(* CoDeSys 2.3.9.48 project: Hausautomation.pro *)
(* Libraries: WagoBuilding_01.lib 14.9.16 07:36:54, SysLibRtc.lib 8.11.10 11:37:48, Gebaeude_allgemein.lib 16.4.15 11:31:36, SysLibTime.lib 8.11.10 11:37:48, Standard.lib*2.6.14 10:37:46, SYSLIBCALLBACK.LIB 8.11.10 11:37:48, Iecsfc.lib 2.6.14 10:37:46 *)

(* PLC configuration (modules and I/O channels)
KA01_KL01_DI AT %IX0.0 [BOOLOnX_I] 1: Flur OG 1 (unten) (Dach 2)
KA01_KL02_DI AT %IX0.1 [BOOLOnX_I] 2: Treppe EG 1
KA02_KL01_DI AT %IX0.2 [BOOLOnX_I] 3: Büro Tür
KA02_KL02_DI AT %IX0.3 [BOOLOnX_I] 4: Eltern Tür
KA02_KL03_DI AT %IX0.4 [BOOLOnX_I] 5: Kind Tür
KA02_KL04_DI AT %IX0.5 [BOOLOnX_I] 6: Küche Tür
KA02_KL05_DI AT %IX0.6 [BOOLOnX_I] 7: WZ Flurtür 1
KA02_KL06_DI AT %IX0.7 [BOOLOnX_I] 8: WZ Terassentür 1
KA02_KL07_DI AT %IX0.8 [BOOLOnX_I] 9: WZ Flurtür 2
KA02_KL08_DI AT %IX0.9 [BOOLOnX_I] 10: Flur Tür WZ
0750-0430 8 DI 24 V DC 3.0ms [Type_1_8_Channels] node 2, in %IX0.2 out %QB0 {INTTypePAAssignment = PLC; INTTypeModule = plugged}
  KA03_KL01_DI AT %IX0.10 [BOOLOnX_I] 11: WZ groß up
  KA03_KL02_DI AT %IX0.11 [BOOLOnX_I] 12: WZ groß: down
  KA03_KL03_DI AT %IX0.12 [BOOLOnX_I] 13: WZ klein up
  KA03_KL04_DI AT %IX0.13 [BOOLOnX_I] 14: WZ klein down
  KA03_KL05_DI AT %IX0.14 [BOOLOnX_I] 15: Kind up
  KA03_KL06_DI AT %IX0.15 [BOOLOnX_I] 16: Kind down
  KA03_KL07_DI AT %IX1.0 [BOOLOnX_I] 17: WZ Tür up
  KA03_KL08_DI AT %IX1.1 [BOOLOnX_I] 18: WZ Tür down
  KA04_KL01_DI AT %IX1.2 [BOOLOnX_I] 19: Eltern down
  KA04_KL02_DI AT %IX1.3 [BOOLOnX_I] 20: Eltern up
  KA04_KL03_DI AT %IX1.4 [BOOLOnX_I] 21: Treppe EG 2
  KA04_KL04_DI AT %IX1.5 [BOOLOnX_I] 22: Haustür
  KA04_KL05_DI AT %IX1.6 [BOOLOnX_I] 23: Flur OG 2 (oben) (Dach 2)
  KA04_KL06_DI AT %IX1.7 [BOOLOnX_I] 24: WZ Flurtür2
  KA04_KL07_DI AT %IX1.8 [BOOLOnX_I] 25: Wand WZ
  KA04_KL08_DI AT %IX1.9 [BOOLOnX_I] 26: Dach Taster 1
KA05_KL01_DO AT %QX0.0 [BOOLOnX_Q] 1: Flur OG
KA05_KL02_DO AT %QX0.1 [BOOLOnX_Q] 2: Flur EG
KA06_KL01_DO AT %QX0.2 [BOOLOnX_Q] 3: Büro
KA06_KL02_DO AT %QX0.3 [BOOLOnX_Q] 4: Eltern
KA06_KL03_DO AT %QX0.4 [BOOLOnX_Q] 5: Kind
KA06_KL04_DO AT %QX0.5 [BOOLOnX_Q] 6: Küche
KA06_KL05_DO AT %QX0.6 [BOOLOnX_Q] 7: WZ 1
KA06_KL06_DO AT %QX0.7 [BOOLOnX_Q] 8: WZ 2
KA06_KL07_DO AT %QX0.8 [BOOLOnX_Q] 9: Essecke Steckdose 1
KA06_KL08_DO AT %QX0.9 [BOOLOnX_Q] 10: Essecke Steckdose 2
KA07_KL01_DO AT %QX0.10 [BOOLOnX_Q] 11: WZ groß down
KA07_KL02_DO AT %QX0.11 [BOOLOnX_Q] 12: WZ groß up
KA07_KL03_DO AT %QX0.12 [BOOLOnX_Q] 13: WZ klein up
KA07_KL04_DO AT %QX0.13 [BOOLOnX_Q] 14: WZ klein down
KA07_KL05_DO AT %QX0.14 [BOOLOnX_Q] 15: Kind down
KA07_KL06_DO AT %QX0.15 [BOOLOnX_Q] 16: Kind up
KA07_KL07_DO AT %QX1.0 [BOOLOnX_Q] 17: Eltern up
KA07_KL08_DO AT %QX1.1 [BOOLOnX_Q] 18: Eltern down
KA08_KL01_DO AT %QX1.2 [BOOLOnX_Q] 19: WZ Tür down
KA08_KL02_DO AT %QX1.3 [BOOLOnX_Q] 20: WZ Tür up
KA08_KL03_DO AT %QX1.4 [BOOLOnX_Q] 21: Dach Lampe 1
KA08_KL04_DO AT %QX1.5 [BOOLOnX_Q] 22: Treppenhaus OG LEDs
KA08_KL05_DO AT %QX1.6 [BOOLOnX_Q] 23: -
KA08_KL06_DO AT %QX1.7 [BOOLOnX_Q] 24: -
KA08_KL07_DO AT %QX1.8 [BOOLOnX_Q] 25: Dach Licht 1
KA08_KL08_DO AT %QX1.9 [BOOLOnX_Q] 26: Dach Licht 2
KA09_KL01_DI AT %IX1.10 [BOOLOnX_I] 27: WZ Terassentür 2
KA09_KL02_DI AT %IX1.11 [BOOLOnX_I] 28: WZ Terassentür 3
KA09_KL03_DI AT %IX1.12 [BOOLOnX_I] 29: WZ Terassentür 4
KA09_KL04_DI AT %IX1.13 [BOOLOnX_I] 30: Büro Up
KA09_KL05_DI AT %IX1.14 [BOOLOnX_I] 31: Büro Down
KA09_KL06_DI AT %IX1.15 [BOOLOnX_I] 32: Küche Down
KA09_KL07_DI AT %IX2.0 [BOOLOnX_I] 33: Küche Up
KA09_KL08_DI AT %IX2.1 [BOOLOnX_I] 34: Dach Taster 2
KA10_KL01_DO AT %QX1.10 [BOOLOnX_Q] 35: Küche Down
KA10_KL02_DO AT %QX1.11 [BOOLOnX_Q] 36: Büro Up
KA10_KL03_DO AT %QX1.12 [BOOLOnX_Q] 37: Büro Down
KA10_KL04_DO AT %QX1.13 [BOOLOnX_Q] 38: Küche Up
KA10_KL05_DO AT %QX1.14 [BOOLOnX_Q] Ch_5 Digital output
KA10_KL06_DO AT %QX1.15 [BOOLOnX_Q] Ch_6 Digital output
KA10_KL07_DO AT %QX2.0 [BOOLOnX_Q] Ch_7 Digital output
KA10_KL08_DO AT %QX2.1 [BOOLOnX_Q] Ch_8 Digital output
KA10_KL09_DO AT %QX2.2 [BOOLOnX_Q] Ch_9 Digital output
KA10_KL10_DO AT %QX2.3 [BOOLOnX_Q] Ch_10 Digital output
KA10_KL11_DO AT %QX2.4 [BOOLOnX_Q] Ch_11 Digital output
KA10_KL12_DO AT %QX2.5 [BOOLOnX_Q] Ch_12 Digital output
KA10_KL13_DO AT %QX2.6 [BOOLOnX_Q] Ch_13 Digital output
KA10_KL14_DO AT %QX2.7 [BOOLOnX_Q] Ch_14 Digital output
KA10_KL15_DO AT %QX2.8 [BOOLOnX_Q] Ch_15 Digital output
KA10_KL16_DO AT %QX2.9 [BOOLOnX_Q] Ch_16 Digital output
Fieldbus variables [FB_VARS] node 1, in %IB0 out %QB0
BOOL, Flag [FLAG_BOOL] node 1, in %IB0 out %QB0
  LichtFlurEG AT %MX0.0 [BOOLOnX_Q] LichtFlurEG(Ausgang)
BOOL, Flag [FLAG_BOOL] node 2, in %IB0 out %QB0
  LichtWohnzimmer AT %MX0.1 [BOOLOnX_Q] LichtWohnzimmer(Ausgang)
BOOL, Flag [FLAG_BOOL] node 3, in %IB0 out %QB0
  LichtKueche AT %MX0.2 [BOOLOnX_Q] LichtKueche(Ausgang)
BOOL, Flag [FLAG_BOOL] node 4, in %IB0 out %QB0
  LichtStehlampe AT %MX0.3 [BOOLOnX_Q] LichtStehlampe(Ausgang)
BOOL, Flag [FLAG_BOOL] node 5, in %IB0 out %QB0
  LichtBuero AT %MX0.4 [BOOLOnX_Q] LichtBuero(Ausgang)
BOOL, Flag [FLAG_BOOL] node 6, in %IB0 out %QB0
  LichtSchlafzimmer AT %MX0.5 [BOOLOnX_Q] LichtSchlafzimmer(Ausgang)
BOOL, Flag [FLAG_BOOL] node 7, in %IB0 out %QB0
  LichtAnnika AT %MX0.6 [BOOLOnX_Q] LichtAnnika(Ausgang)
BOOL, Flag [FLAG_BOOL] node 8, in %IB0 out %QB0
  LichtFlurOG AT %MX0.7 [BOOLOnX_Q] LichtFlurOG(Ausgang)
BOOL, Flag [FLAG_BOOL] node 9, in %IB0 out %QB0
  TasterBuero AT %MX0.8 [BOOLOnX_Q] TasterBuero(Eingang)
BOOL, Flag [FLAG_BOOL] node 10, in %IB0 out %QB0
  TasterFlurEG AT %MX0.9 [BOOLOnX_Q] TasterFlurEG(Eingang)
BOOL, Flag [FLAG_BOOL] node 11, in %IB0 out %QB0
  TasterWohnzimmer AT %MX0.10 [BOOLOnX_Q] TasterWohnzimmer(Eingang)
BOOL, Flag [FLAG_BOOL] node 12, in %IB0 out %QB0
  TasterKueche AT %MX0.11 [BOOLOnX_Q] TasterKueche(Eingang)
BOOL, Flag [FLAG_BOOL] node 13, in %IB0 out %QB0
  TasterStehlampe AT %MX0.12 [BOOLOnX_Q] TasterStehlampe(Eingang)
BOOL, Flag [FLAG_BOOL] node 14, in %IB0 out %QB0
  TasterSchlafzimmer AT %MX0.13 [BOOLOnX_Q] TasterSchlafzimmer(Eingang)
BOOL, Flag [FLAG_BOOL] node 15, in %IB0 out %QB0
  TasterAnnika AT %MX0.14 [BOOLOnX_Q] TasterAnnika(Eingang)
BOOL, Flag [FLAG_BOOL] node 16, in %IB0 out %QB0
  TasterFlurOG AT %MX0.15 [BOOLOnX_Q] TasterFlurOG(Eingang)
BOOL, Flag [FLAG_BOOL] node 17, in %IB0 out %QB0
  JalousieElternUp AT %MX1.0 [BOOLOnX_Q] Jalousie Eltern Hoch
BOOL, Flag [FLAG_BOOL] node 18, in %IB0 out %QB0
  JalousieElternDown AT %MX1.1 [BOOLOnX_Q] Jalousie Eltern Runter
BOOL, Flag [FLAG_BOOL] node 19, in %IB0 out %QB0
  JalousieAnnikaDown AT %MX1.2 [BOOLOnX_Q] Jalousie Annika runter
BOOL, Flag [FLAG_BOOL] node 20, in %IB0 out %QB0
  JalousieAnnikaUp AT %MX1.3 [BOOLOnX_Q] Jalousie Annika hoch
BOOL, Flag [FLAG_BOOL] node 21, in %IB0 out %QB0
  JalousieWohnzimmerGrossDown AT %MX1.4 [BOOLOnX_Q] Jalousie Wohnzimmer großes Fenster runter
BOOL, Flag [FLAG_BOOL] node 22, in %IB0 out %QB0
  JalousieWohnzimmerGrossUp AT %MX1.5 [BOOLOnX_Q] Jalousie Wohnzimmer großes Fenster hoch
BOOL, Flag [FLAG_BOOL] node 23, in %IB0 out %QB0
  JalousieWohnzimmerTuerDown AT %MX1.6 [BOOLOnX_Q] Jalousie Wohnzimmer Tür runter
BOOL, Flag [FLAG_BOOL] node 24, in %IB0 out %QB0
  JalousieWohnzimmerTuerUp AT %MX1.7 [BOOLOnX_Q] Jalousie Wohnzimmer Tür hoch
BOOL, Flag [FLAG_BOOL] node 25, in %IB0 out %QB0
  JalousieWohnzimmerKleinDown AT %MX1.8 [BOOLOnX_Q] Jalousie Wohnzimmer kleines Fenster runter
BOOL, Flag [FLAG_BOOL] node 26, in %IB0 out %QB0
  JalousieWohnzimmerKleinUp AT %MX1.9 [BOOLOnX_Q] Jalousie Wohnzimmer kleines Fenster hoch
BOOL, Flag [FLAG_BOOL] node 27, in %IB0 out %QB0
  JalousieBueroUp AT %MX1.10 [BOOLOnX_Q] Jalousie Büro hoch
BOOL, Flag [FLAG_BOOL] node 28, in %IB0 out %QB0
  JalousieBueroDown AT %MX1.11 [BOOLOnX_Q] Jalousie Büro runter
BOOL, Flag [FLAG_BOOL] node 29, in %IB0 out %QB0
  JalousieKuecheUp AT %MX1.12 [BOOLOnX_Q] Jalousie Küche hoch
BOOL, Flag [FLAG_BOOL] node 30, in %IB0 out %QB0
  JalousieKuecheDown AT %MX1.13 [BOOLOnX_Q] Jalousie Küche runter
BOOL, Flag [FLAG_BOOL] node 31, in %IB0 out %QB0
  TasterLichtDachboden AT %MX1.14 [BOOLOnX_Q] Taster Licht Dachboden
BOOL, Flag [FLAG_BOOL] node 32, in %IB0 out %QB0
  LichtDachbodenVorne AT %MX1.15 [BOOLOnX_Q] Licht Dachboden vorne (Büro)
BOOL, Flag [FLAG_BOOL] node 33, in %IB0 out %QB0
  LichtDachbodenHinten AT %MX2.0 [BOOLOnX_Q] Licht Dachboden hinten (Gästezimmer)
Modbus-Master [MB_MASTER] node 3, in %IB0 out %QB0
*)

(* Task configuration *)
TASK MAIN (PRIORITY := 1, INTERVAL := T#200ms);
	PLC_PRG();
END_TASK

(* Global variable list: Globale_Variablen *)
VAR_GLOBAL

	LIGHT_CentralOn: BOOL := FALSE;
	LIGHT_CentralOff: BOOL := FALSE;
	WZ_2_AN: BOOL;

	YEAR: WORD;
	MONTH: BYTE;
	DAY: BYTE;
	HOUR: BYTE;
	MINUTE: BYTE;
	SECOND: BYTE;
	WEEK_DAY: BYTE;


      DAY_BOOL: BOOL;
      NIGHT_BOOL: BOOL;

	BLINDS_CentralUp: BOOL := FALSE;
	BLINDS_LfzGesamt: UINT := 700;
	BLINDS_PauseAufAb: UINT := 5;
	BLINDS_TasKurz: UINT := 5;
	BLINDS_LfzBeschattPos: UINT := 10;
	BLINDS_LfzKurz: UINT := 400;
	BLINDS_WendeZeitLamelle: UINT := 40;
END_VAR

(* POU PLC_PRG, ST *)
PROGRAM PLC_PRG
LIGHTS_FLUR_EG;
LIGHTS_FLUR_OG;
LIGHTS_WZ;
LIGHTS_KUECHE;
LIGHTS_BUERO;
LIGHTS_SCHLAFZIMMER;
LIGHTS_ANNIKA;
LIGHTS_STEHLAMPE;
LIGHTS_DRAUSSEN;
UHRZEIT;
BLINDS_WZ;
BLINDS_ANNIKA;
BLINDS_ELTERN;
BLINDS_BUERO;
BLINDS_KUECHE;
LIGHTS_ATTIC;
IsDay;
END_PROGRAM

(* POU LIGHTS_FLUR_EG, CFC *)
PROGRAM LIGHTS_FLUR_EG
VAR
	FB_LIGHT_02: FbLatchedRelay;
	F_Treppe_1: F_TRIG;
	F_Treppe_2: R_TRIG;
	FB_LIGHT_02_2: FbLatchedRelay;
	F_Haustuer_1: F_TRIG;
	F_Haustuer_2: R_TRIG;
	F_FlurTuerWZ_1: F_TRIG;
	F_FlurTuerWZ_2: R_TRIG;
	F_Flur_oben_1: F_TRIG;
	F_Flur_oben_2: R_TRIG;
	F_Flur_OG_1: F_TRIG;
	F_Flur_OG_2: R_TRIG;
	F_Flur_EG_5: F_TRIG;
	F_Flur_EG_6: R_TRIG;
	F_Flur_EG_openhab: F_TRIG;
	F_Flur_openhab: R_TRIG;
	R_Flur_EG_openhab: R_TRIG;
END_VAR
VAR (* helpers for the ST form of the networks *)
	_t138 : BOOL;
END_VAR
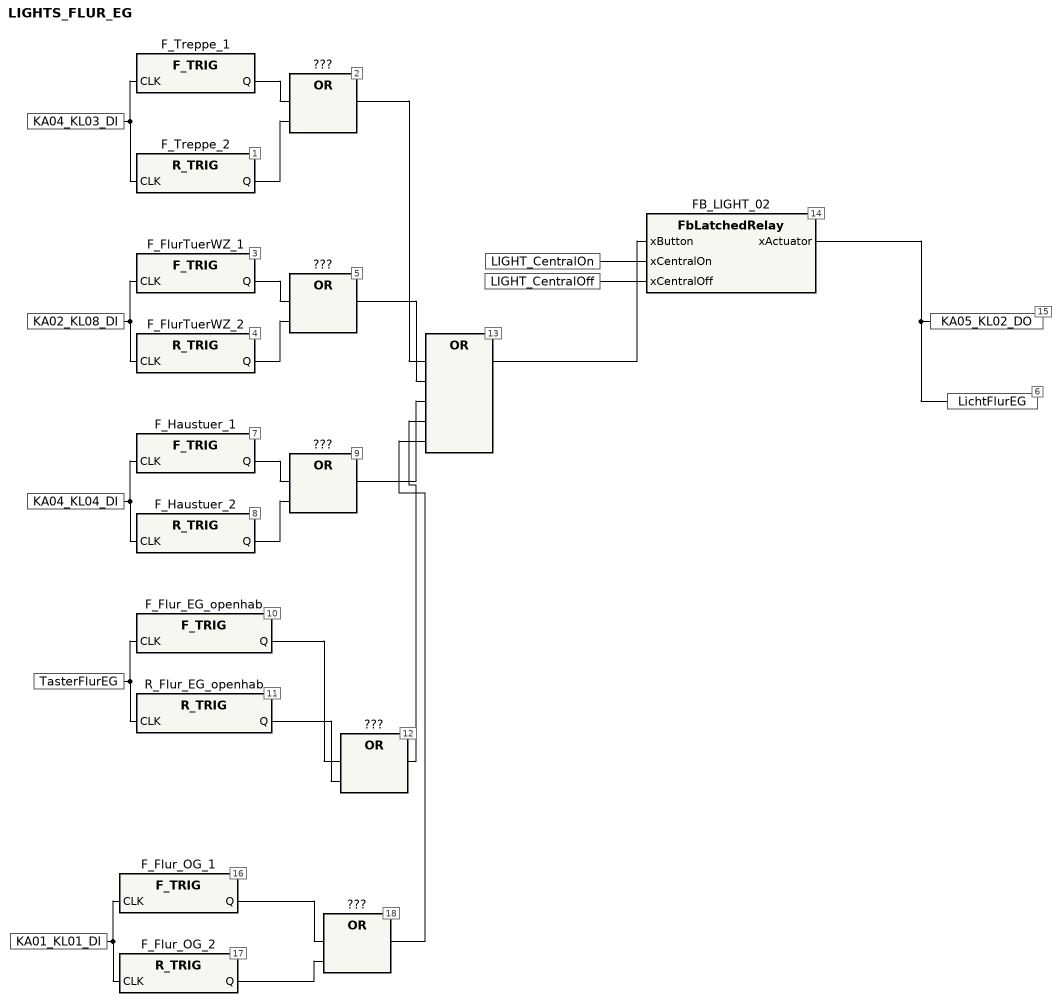
_CFC_ (* Continuous Function Chart, elements in execution order *)
#0 F_Treppe_1:F_TRIG(CLK: KA04_KL03_DI)
#1 F_Treppe_2:R_TRIG(CLK: KA04_KL03_DI)
#2 ???:OR(#0.Q, #1.Q)
#3 F_FlurTuerWZ_1:F_TRIG(CLK: KA02_KL08_DI)
#4 F_FlurTuerWZ_2:R_TRIG(CLK: KA02_KL08_DI)
#5 ???:OR(#3.Q, #4.Q)
#6 LichtFlurEG <= #14.xActuator
#7 F_Haustuer_1:F_TRIG(CLK: KA04_KL04_DI)
#8 F_Haustuer_2:R_TRIG(CLK: KA04_KL04_DI)
#9 ???:OR(#7.Q, #8.Q)
#10 F_Flur_EG_openhab:F_TRIG(CLK: TasterFlurEG)
#11 R_Flur_EG_openhab:R_TRIG(CLK: TasterFlurEG)
#12 ???:OR(#10.Q, #11.Q)
#13 OR(#2, #5, #9, #12, #18)
#14 FB_LIGHT_02:FbLatchedRelay(xButton: #13, xCentralOn: LIGHT_CentralOn, xCentralOff: LIGHT_CentralOff)
#15 KA05_KL02_DO <= #14.xActuator
#16 F_Flur_OG_1:F_TRIG(CLK: KA01_KL01_DI)
#17 F_Flur_OG_2:R_TRIG(CLK: KA01_KL01_DI)
#18 ???:OR(#16.Q, #17.Q)
_END_CFC_
(* the same logic as Structured Text *)
F_Treppe_1(CLK := KA04_KL03_DI);
F_Treppe_2(CLK := KA04_KL03_DI);
F_FlurTuerWZ_1(CLK := KA02_KL08_DI);
F_FlurTuerWZ_2(CLK := KA02_KL08_DI);
LichtFlurEG := FB_LIGHT_02.xActuator;
F_Haustuer_1(CLK := KA04_KL04_DI);
F_Haustuer_2(CLK := KA04_KL04_DI);
F_Flur_EG_openhab(CLK := TasterFlurEG);
R_Flur_EG_openhab(CLK := TasterFlurEG);
FB_LIGHT_02(xButton := (F_Treppe_1.Q OR F_Treppe_2.Q) OR (F_FlurTuerWZ_1.Q OR F_FlurTuerWZ_2.Q) OR (F_Haustuer_1.Q OR F_Haustuer_2.Q) OR (F_Flur_EG_openhab.Q OR R_Flur_EG_openhab.Q) OR _t138, xCentralOn := LIGHT_CentralOn, xCentralOff := LIGHT_CentralOff);
KA05_KL02_DO := FB_LIGHT_02.xActuator;
F_Flur_OG_1(CLK := KA01_KL01_DI);
F_Flur_OG_2(CLK := KA01_KL01_DI);
_t138 := F_Flur_OG_1.Q OR F_Flur_OG_2.Q;
END_PROGRAM

(* POU LIGHTS_FLUR_OG, CFC *)
PROGRAM LIGHTS_FLUR_OG
VAR
	FB_LIGHT_01: FbLatchedRelay;
	F_FLUR_EG_OBEN_1: F_TRIG;
	F_FLUR_EG_OBEN_2: R_TRIG;
	F_FLUR_OBEN_1: F_TRIG;
	F_FLUR_OBEN_3: R_TRIG;
	T_Licht_LEDs: TON;
	RS_LEDs: RS;
	F_FLUR_OBEN_openhab: F_TRIG;
	R_FLUR_OBEN_openhab: R_TRIG;
	Fb_Klick_OG: Fb_Klick;
	FB_LIGHT_02: FbLatchedRelay;
	R_TRIG_DACHBODEN2_openhab: R_TRIG;
      F_TRIG_DACHBODEN2_openhab: F_TRIG;

	F_FLUR_OG_OBEN_1: F_TRIG;
	R_FLUR_OG_OBEN_2: R_TRIG;
END_VAR
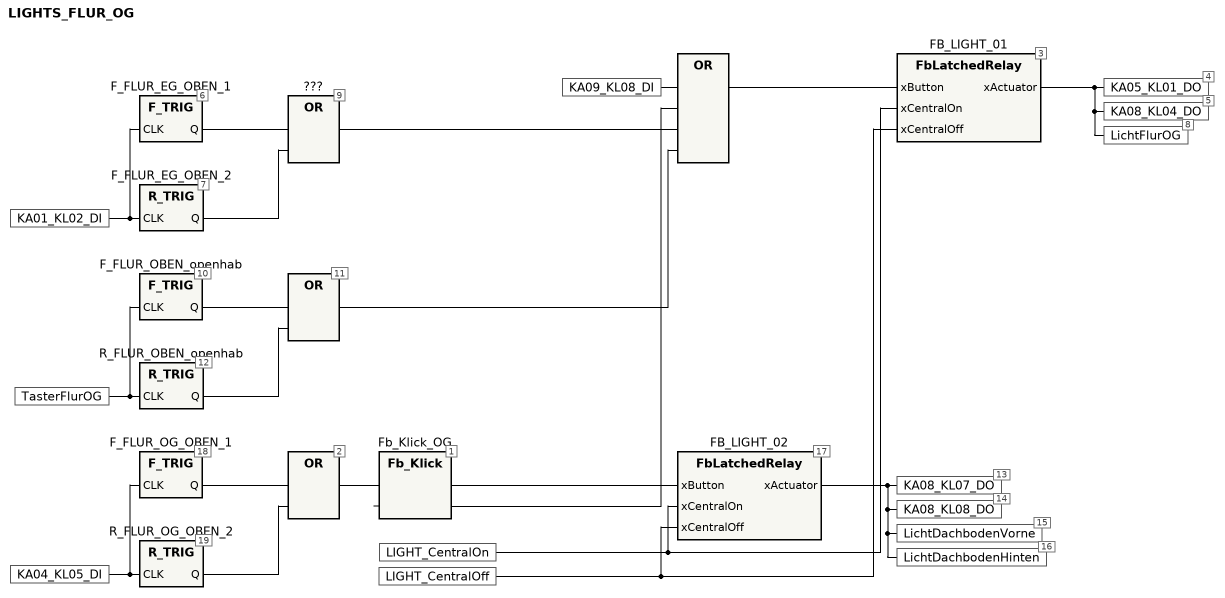
_CFC_ (* Continuous Function Chart, elements in execution order *)
#0 OR(KA09_KL08_DI, #1.out 2, #9, #11)
#1 Fb_Klick_OG:Fb_Klick(#2, -)
#2 OR(#18.Q, #19.Q)
#3 FB_LIGHT_01:FbLatchedRelay(xButton: #0, xCentralOn: LIGHT_CentralOn, xCentralOff: LIGHT_CentralOff)
#4 KA05_KL01_DO <= #3.xActuator
#5 KA08_KL04_DO <= #3.xActuator
#6 F_FLUR_EG_OBEN_1:F_TRIG(CLK: KA01_KL02_DI)
#7 F_FLUR_EG_OBEN_2:R_TRIG(CLK: KA01_KL02_DI)
#8 LichtFlurOG <= #3.xActuator
#9 ???:OR(#6.Q, #7.Q)
#10 F_FLUR_OBEN_openhab:F_TRIG(CLK: TasterFlurOG)
#11 OR(#10.Q, #12.Q)
#12 R_FLUR_OBEN_openhab:R_TRIG(CLK: TasterFlurOG)
#13 KA08_KL07_DO <= #17.xActuator
#14 KA08_KL08_DO <= #17.xActuator
#15 LichtDachbodenVorne <= #17.xActuator
#16 LichtDachbodenHinten <= #17.xActuator
#17 FB_LIGHT_02:FbLatchedRelay(xButton: #1.out 1, xCentralOn: LIGHT_CentralOn, xCentralOff: LIGHT_CentralOff)
#18 F_FLUR_OG_OBEN_1:F_TRIG(CLK: KA04_KL05_DI)
#19 R_FLUR_OG_OBEN_2:R_TRIG(CLK: KA04_KL05_DI)
_END_CFC_
END_PROGRAM

(* POU LIGHTS_WZ, CFC *)
PROGRAM LIGHTS_WZ
VAR

	R_TRIG_ESS_1: R_TRIG;

	R_TRIG_ESS1: R_TRIG;
	F_TRIG_ESS1: F_TRIG;
	FB_LIGHT_07: FbLatchedRelay;
	FB_LIGHT_08: FbLatchedRelay;
	FB_LIGHT_09: FbLatchedRelay;
	FB_LIGHT_10: FbLatchedRelay;
	R_TRIB_WZ_1: R_TRIG;
	F_TRIG_WZ_2: F_TRIG;
	R_TRIG_WZ_3: R_TRIG;
	F_TRIG_WZ_4: F_TRIG;
	WZ_1_AN: BOOL;
	KA08_KL05_DA: BOOL;
	R_TRIG_DRAUSSEN: R_TRIG;
	F_TRIG_DRAUSSEN: F_TRIG;

	R_TRIG_WZ_openhab: R_TRIG;
	F_TRIG_WZ_openhab: F_TRIG;


	R_TRIG_STEHLAMPE_openhab: R_TRIG;
	F_TRIG_STEHLAMPE_openhab: F_TRIG;
	FB_KLICK_Taster: Fb_Klick;
	R_TRIG_WZ_3_openhab: R_TRIG;
	F_TRIG_WZ_3_openhab: F_TRIG;
END_VAR
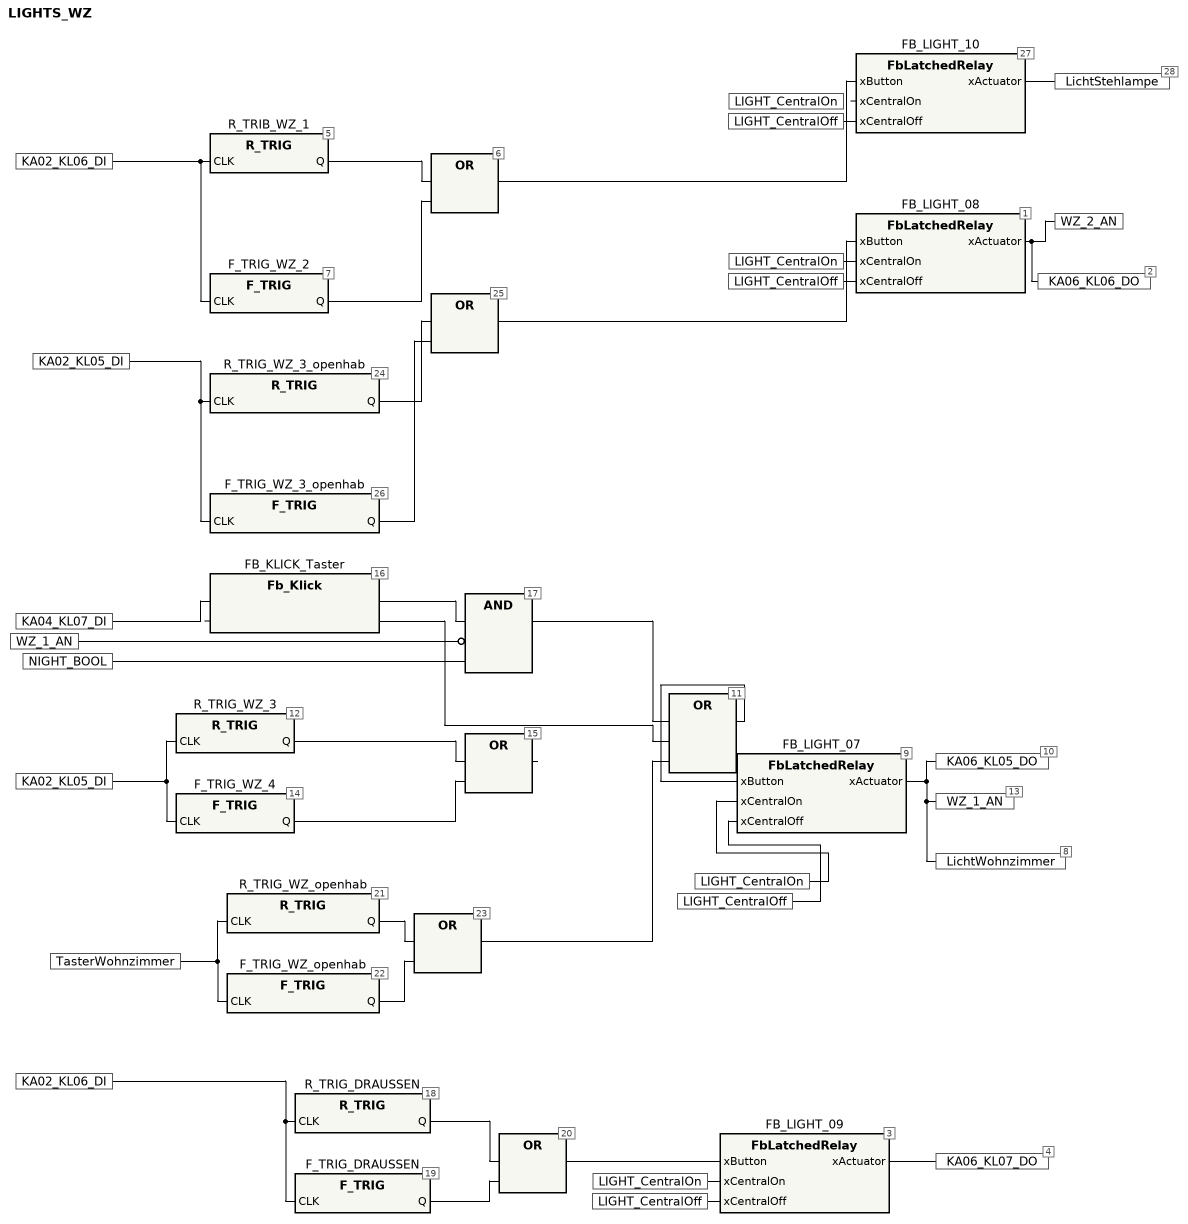
_CFC_ (* Continuous Function Chart, elements in execution order *)
#0 WZ_2_AN <= #1.xActuator
#1 FB_LIGHT_08:FbLatchedRelay(xButton: #25, xCentralOn: LIGHT_CentralOn, xCentralOff: LIGHT_CentralOff)
#2 KA06_KL06_DO <= #1.xActuator
#3 FB_LIGHT_09:FbLatchedRelay(xButton: #20, xCentralOn: LIGHT_CentralOn, xCentralOff: LIGHT_CentralOff)
#4 KA06_KL07_DO <= #3.xActuator
#5 R_TRIB_WZ_1:R_TRIG(CLK: KA02_KL06_DI)
#6 OR(#5.Q, #7.Q)
#7 F_TRIG_WZ_2:F_TRIG(CLK: KA02_KL06_DI)
#8 LichtWohnzimmer <= #9.xActuator
#9 FB_LIGHT_07:FbLatchedRelay(xButton: #11, xCentralOn: LIGHT_CentralOn, xCentralOff: LIGHT_CentralOff)
#10 KA06_KL05_DO <= #9.xActuator
#11 OR(#17, #16.out 2, #23)
#12 R_TRIG_WZ_3:R_TRIG(CLK: KA02_KL05_DI)
#13 WZ_1_AN <= #9.xActuator
#14 F_TRIG_WZ_4:F_TRIG(CLK: KA02_KL05_DI)
#15 OR(#12.Q, #14.Q)
#16 FB_KLICK_Taster:Fb_Klick(KA04_KL07_DI, -)
#17 AND(#16.out 1, NOT WZ_1_AN, NIGHT_BOOL)
#18 R_TRIG_DRAUSSEN:R_TRIG(CLK: KA02_KL06_DI)
#19 F_TRIG_DRAUSSEN:F_TRIG(CLK: KA02_KL06_DI)
#20 OR(#18.Q, #19.Q)
#21 R_TRIG_WZ_openhab:R_TRIG(CLK: TasterWohnzimmer)
#22 F_TRIG_WZ_openhab:F_TRIG(CLK: TasterWohnzimmer)
#23 OR(#21.Q, #22.Q)
#24 R_TRIG_WZ_3_openhab:R_TRIG(CLK: KA02_KL05_DI)
#25 OR(#24.Q, #26.Q)
#26 F_TRIG_WZ_3_openhab:F_TRIG(CLK: KA02_KL05_DI)
unconnected input LIGHT_CentralOn
#27 FB_LIGHT_10:FbLatchedRelay(xButton: #6, xCentralOn: -, xCentralOff: LIGHT_CentralOff)
#28 LichtStehlampe <= #27.xActuator
_END_CFC_
END_PROGRAM

(* POU LIGHTS_KUECHE, CFC *)
PROGRAM LIGHTS_KUECHE
VAR
	R_TRIG_KUECHE1: R_TRIG;
	F_TRIG_KUECHE2: F_TRIG;
	FB_LIGHT_06: FbLatchedRelay;
	R_TRIG_KUECHE1_openhab: R_TRIG;
	F_TRIG_KUECHE2_openhab: F_TRIG;
END_VAR
VAR (* helpers for the ST form of the networks *)
	_t15 : BOOL;
	_t24 : BOOL;
END_VAR
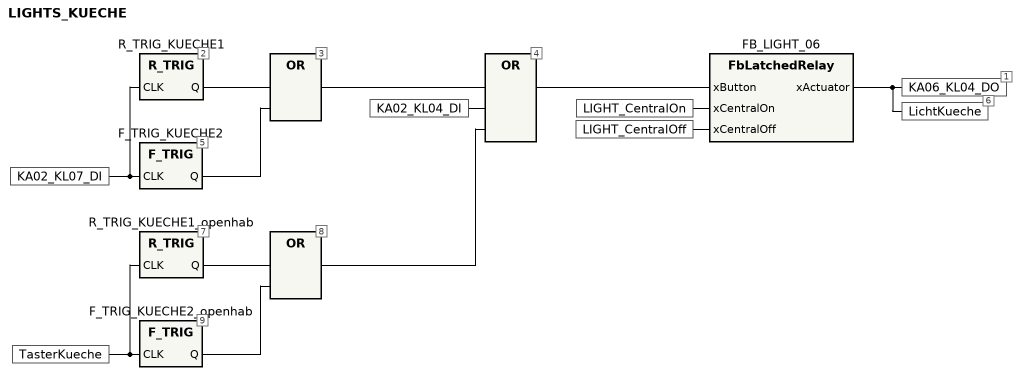
_CFC_ (* Continuous Function Chart, elements in execution order *)
#0 FB_LIGHT_06:FbLatchedRelay(xButton: #4, xCentralOn: LIGHT_CentralOn, xCentralOff: LIGHT_CentralOff)
#1 KA06_KL04_DO <= #0.xActuator
#2 R_TRIG_KUECHE1:R_TRIG(CLK: KA02_KL07_DI)
#3 OR(#2.Q, #5.Q)
#4 OR(#3, KA02_KL04_DI, #8)
#5 F_TRIG_KUECHE2:F_TRIG(CLK: KA02_KL07_DI)
#6 LichtKueche <= #0.xActuator
#7 R_TRIG_KUECHE1_openhab:R_TRIG(CLK: TasterKueche)
#8 OR(#7.Q, #9.Q)
#9 F_TRIG_KUECHE2_openhab:F_TRIG(CLK: TasterKueche)
_END_CFC_
(* the same logic as Structured Text *)
FB_LIGHT_06(xButton := _t15, xCentralOn := LIGHT_CentralOn, xCentralOff := LIGHT_CentralOff);
KA06_KL04_DO := FB_LIGHT_06.xActuator;
R_TRIG_KUECHE1(CLK := KA02_KL07_DI);
_t15 := (R_TRIG_KUECHE1.Q OR F_TRIG_KUECHE2.Q) OR KA02_KL04_DI OR _t24;
F_TRIG_KUECHE2(CLK := KA02_KL07_DI);
LichtKueche := FB_LIGHT_06.xActuator;
R_TRIG_KUECHE1_openhab(CLK := TasterKueche);
_t24 := R_TRIG_KUECHE1_openhab.Q OR F_TRIG_KUECHE2_openhab.Q;
F_TRIG_KUECHE2_openhab(CLK := TasterKueche);
END_PROGRAM

(* POU LIGHTS_BUERO, CFC *)
PROGRAM LIGHTS_BUERO
VAR

	FB_LIGHT_03: FbLatchedRelay;

	F_TRIG_WZ_1: F_TRIG;
	R_TRIG_WZ_1: R_TRIG;
END_VAR
VAR (* helpers for the ST form of the networks *)
	_t85 : BOOL;
	_t83 : BOOL;
END_VAR
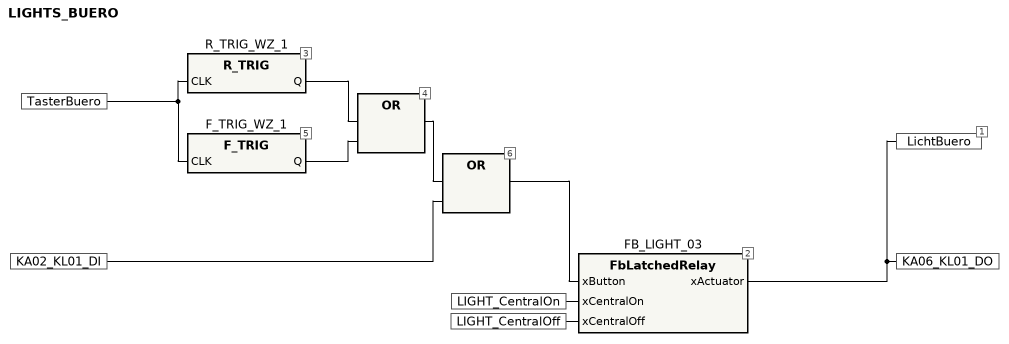
_CFC_ (* Continuous Function Chart, elements in execution order *)
#0 KA06_KL01_DO <= #2.xActuator
#1 LichtBuero <= #2.xActuator
#2 FB_LIGHT_03:FbLatchedRelay(xButton: #6, xCentralOn: LIGHT_CentralOn, xCentralOff: LIGHT_CentralOff)
#3 R_TRIG_WZ_1:R_TRIG(CLK: TasterBuero)
#4 OR(#3.Q, #5.Q)
#5 F_TRIG_WZ_1:F_TRIG(CLK: TasterBuero)
#6 OR(#4, KA02_KL01_DI)
_END_CFC_
(* the same logic as Structured Text *)
KA06_KL01_DO := FB_LIGHT_03.xActuator;
LichtBuero := FB_LIGHT_03.xActuator;
FB_LIGHT_03(xButton := _t85, xCentralOn := LIGHT_CentralOn, xCentralOff := LIGHT_CentralOff);
R_TRIG_WZ_1(CLK := TasterBuero);
_t83 := R_TRIG_WZ_1.Q OR F_TRIG_WZ_1.Q;
F_TRIG_WZ_1(CLK := TasterBuero);
_t85 := _t83 OR KA02_KL01_DI;
END_PROGRAM

(* POU LIGHTS_SCHLAFZIMMER, CFC *)
PROGRAM LIGHTS_SCHLAFZIMMER
VAR

	FB_LIGHT_04: FbLatchedRelay;

	R_TRIG_SCHLAZIMMER_openhab: R_TRIG;
	F_TRIG_SCHLAFZIMMER_openhab: F_TRIG;
END_VAR
VAR (* helpers for the ST form of the networks *)
	_t64 : BOOL;
END_VAR
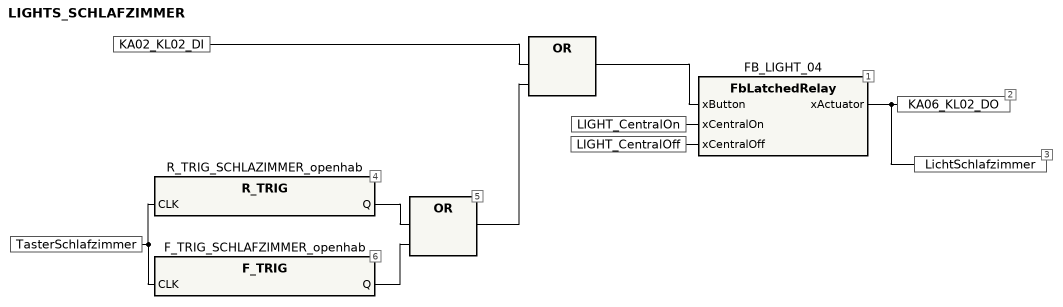
_CFC_ (* Continuous Function Chart, elements in execution order *)
#0 OR(KA02_KL02_DI, #5)
#1 FB_LIGHT_04:FbLatchedRelay(xButton: #0, xCentralOn: LIGHT_CentralOn, xCentralOff: LIGHT_CentralOff)
#2 KA06_KL02_DO <= #1.xActuator
#3 LichtSchlafzimmer <= #1.xActuator
#4 R_TRIG_SCHLAZIMMER_openhab:R_TRIG(CLK: TasterSchlafzimmer)
#5 OR(#4.Q, #6.Q)
#6 F_TRIG_SCHLAFZIMMER_openhab:F_TRIG(CLK: TasterSchlafzimmer)
_END_CFC_
(* the same logic as Structured Text *)
FB_LIGHT_04(xButton := KA02_KL02_DI OR _t64, xCentralOn := LIGHT_CentralOn, xCentralOff := LIGHT_CentralOff);
KA06_KL02_DO := FB_LIGHT_04.xActuator;
LichtSchlafzimmer := FB_LIGHT_04.xActuator;
R_TRIG_SCHLAZIMMER_openhab(CLK := TasterSchlafzimmer);
_t64 := R_TRIG_SCHLAZIMMER_openhab.Q OR F_TRIG_SCHLAFZIMMER_openhab.Q;
F_TRIG_SCHLAFZIMMER_openhab(CLK := TasterSchlafzimmer);
END_PROGRAM

(* POU LIGHTS_ANNIKA, CFC *)
PROGRAM LIGHTS_ANNIKA
VAR
	FB_LIGHT_05: FbLatchedRelay;

	R_TRIG_ANNIKA_openhab: R_TRIG;
	F_TRIG_ANNIKA_openhab: F_TRIG;
END_VAR
VAR (* helpers for the ST form of the networks *)
	_t72 : BOOL;
	_t69 : BOOL;
END_VAR
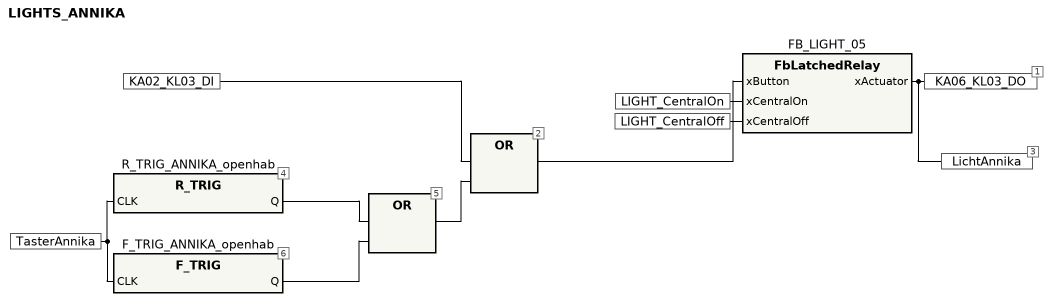
_CFC_ (* Continuous Function Chart, elements in execution order *)
#0 FB_LIGHT_05:FbLatchedRelay(xButton: #2, xCentralOn: LIGHT_CentralOn, xCentralOff: LIGHT_CentralOff)
#1 KA06_KL03_DO <= #0.xActuator
#2 OR(KA02_KL03_DI, #5)
#3 LichtAnnika <= #0.xActuator
#4 R_TRIG_ANNIKA_openhab:R_TRIG(CLK: TasterAnnika)
#5 OR(#4.Q, #6.Q)
#6 F_TRIG_ANNIKA_openhab:F_TRIG(CLK: TasterAnnika)
_END_CFC_
(* the same logic as Structured Text *)
FB_LIGHT_05(xButton := _t72, xCentralOn := LIGHT_CentralOn, xCentralOff := LIGHT_CentralOff);
KA06_KL03_DO := FB_LIGHT_05.xActuator;
_t72 := KA02_KL03_DI OR _t69;
LichtAnnika := FB_LIGHT_05.xActuator;
R_TRIG_ANNIKA_openhab(CLK := TasterAnnika);
_t69 := R_TRIG_ANNIKA_openhab.Q OR F_TRIG_ANNIKA_openhab.Q;
F_TRIG_ANNIKA_openhab(CLK := TasterAnnika);
END_PROGRAM

(* POU LIGHTS_STEHLAMPE, CFC *)
PROGRAM LIGHTS_STEHLAMPE
VAR

	FB_LIGHT_10: FbLatchedRelay;
	LichtSAtehlampe: BOOL;
	R_TRIG_STEHLAMPE_1: R_TRIG;
	F_TRIG_STEHLAMPE_2: F_TRIG;
	R_TRIG_TERASSE_1: R_TRIG;
	F_TRIG_TERASSE_2: F_TRIG;
	R_TRIG_TERASSE_2: R_TRIG;
	F_TRIG_TERASSE_1: F_TRIG;
END_VAR
VAR (* helpers for the ST form of the networks *)
	_t97 : BOOL;
END_VAR
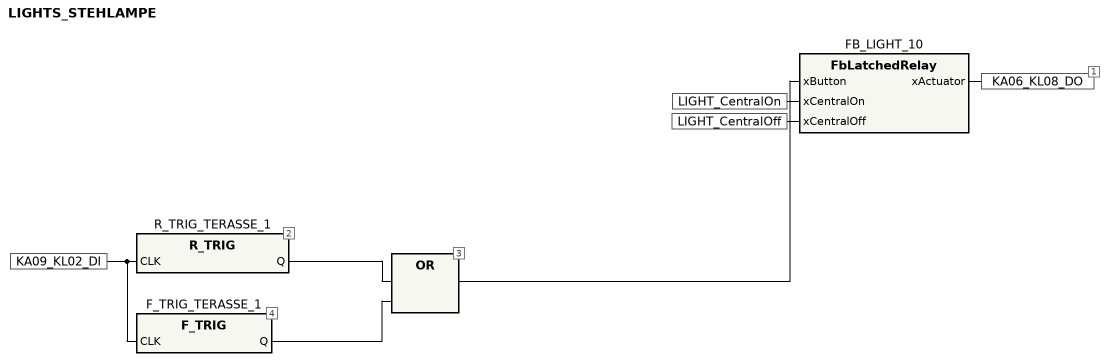
_CFC_ (* Continuous Function Chart, elements in execution order *)
#0 FB_LIGHT_10:FbLatchedRelay(xButton: #3, xCentralOn: LIGHT_CentralOn, xCentralOff: LIGHT_CentralOff)
#1 KA06_KL08_DO <= #0.xActuator
#2 R_TRIG_TERASSE_1:R_TRIG(CLK: KA09_KL02_DI)
#3 OR(#2.Q, #4.Q)
#4 F_TRIG_TERASSE_1:F_TRIG(CLK: KA09_KL02_DI)
_END_CFC_
(* the same logic as Structured Text *)
FB_LIGHT_10(xButton := _t97, xCentralOn := LIGHT_CentralOn, xCentralOff := LIGHT_CentralOff);
KA06_KL08_DO := FB_LIGHT_10.xActuator;
R_TRIG_TERASSE_1(CLK := KA09_KL02_DI);
_t97 := R_TRIG_TERASSE_1.Q OR F_TRIG_TERASSE_1.Q;
F_TRIG_TERASSE_1(CLK := KA09_KL02_DI);
END_PROGRAM

(* POU LIGHTS_DRAUSSEN, CFC *)
PROGRAM LIGHTS_DRAUSSEN
VAR

	R_TRIG_ESS1: R_TRIG;
	F_TRIG_ESS1: F_TRIG;
	FB_LIGHT_10: FbLatchedRelay;

END_VAR
VAR (* helpers for the ST form of the networks *)
	_t324 : BOOL;
END_VAR
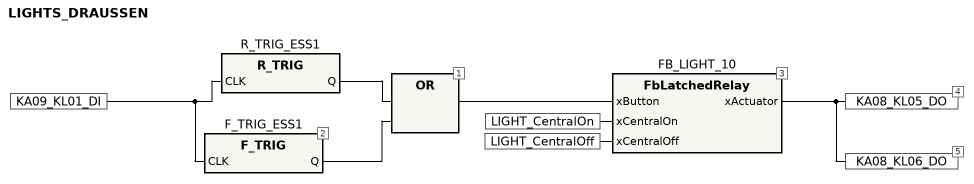
_CFC_ (* Continuous Function Chart, elements in execution order *)
#0 R_TRIG_ESS1:R_TRIG(CLK: KA09_KL01_DI)
#1 OR(#0.Q, #2.Q)
#2 F_TRIG_ESS1:F_TRIG(CLK: KA09_KL01_DI)
#3 FB_LIGHT_10:FbLatchedRelay(xButton: #1, xCentralOn: LIGHT_CentralOn, xCentralOff: LIGHT_CentralOff)
#4 KA08_KL05_DO <= #3.xActuator
#5 KA08_KL06_DO <= #3.xActuator
_END_CFC_
(* the same logic as Structured Text *)
R_TRIG_ESS1(CLK := KA09_KL01_DI);
_t324 := R_TRIG_ESS1.Q OR F_TRIG_ESS1.Q;
F_TRIG_ESS1(CLK := KA09_KL01_DI);
FB_LIGHT_10(xButton := _t324, xCentralOn := LIGHT_CentralOn, xCentralOff := LIGHT_CentralOff);
KA08_KL05_DO := FB_LIGHT_10.xActuator;
KA08_KL06_DO := FB_LIGHT_10.xActuator;
END_PROGRAM

(* POU UHRZEIT, CFC *)
PROGRAM UHRZEIT
VAR
	UHRZEIT: FB_Time;

	VAR_TRUE: BOOL := TRUE;
	in_YEAR: WORD := 2017;
	in_MONTH: BYTE :=4;
	in_DAY: BYTE := 12;
	in_HOUR: BYTE:= 19;
	in_MINUTE: BYTE := 44;
	in_SECOND: BYTE :=0;

END_VAR
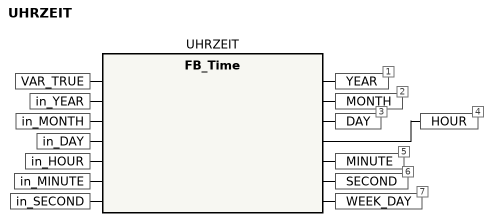
_CFC_ (* Continuous Function Chart, elements in execution order *)
#0 UHRZEIT:FB_Time(VAR_TRUE, in_YEAR, in_MONTH, in_DAY, in_HOUR, in_MINUTE, in_SECOND)
#1 YEAR <= #0.out 1
#2 MONTH <= #0.out 2
#3 DAY <= #0.out 3
#4 HOUR <= #0.out 4
#5 MINUTE <= #0.out 5
#6 SECOND <= #0.out 6
#7 WEEK_DAY <= #0.out 7
_END_CFC_
END_PROGRAM

(* POU BLINDS_WZ, CFC *)
PROGRAM BLINDS_WZ
VAR

	FBJalousie_01: FbJalousie;
	JalPos_01: BYTE;
	FBJalousie_02: FbJalousie;
	JalPos_02: BYTE;
	FBJalousie_05: FbJalousie;
	JalPos_05: BYTE;

	FB_BLINDS_DBKLICK: Fb_Klick;
END_VAR
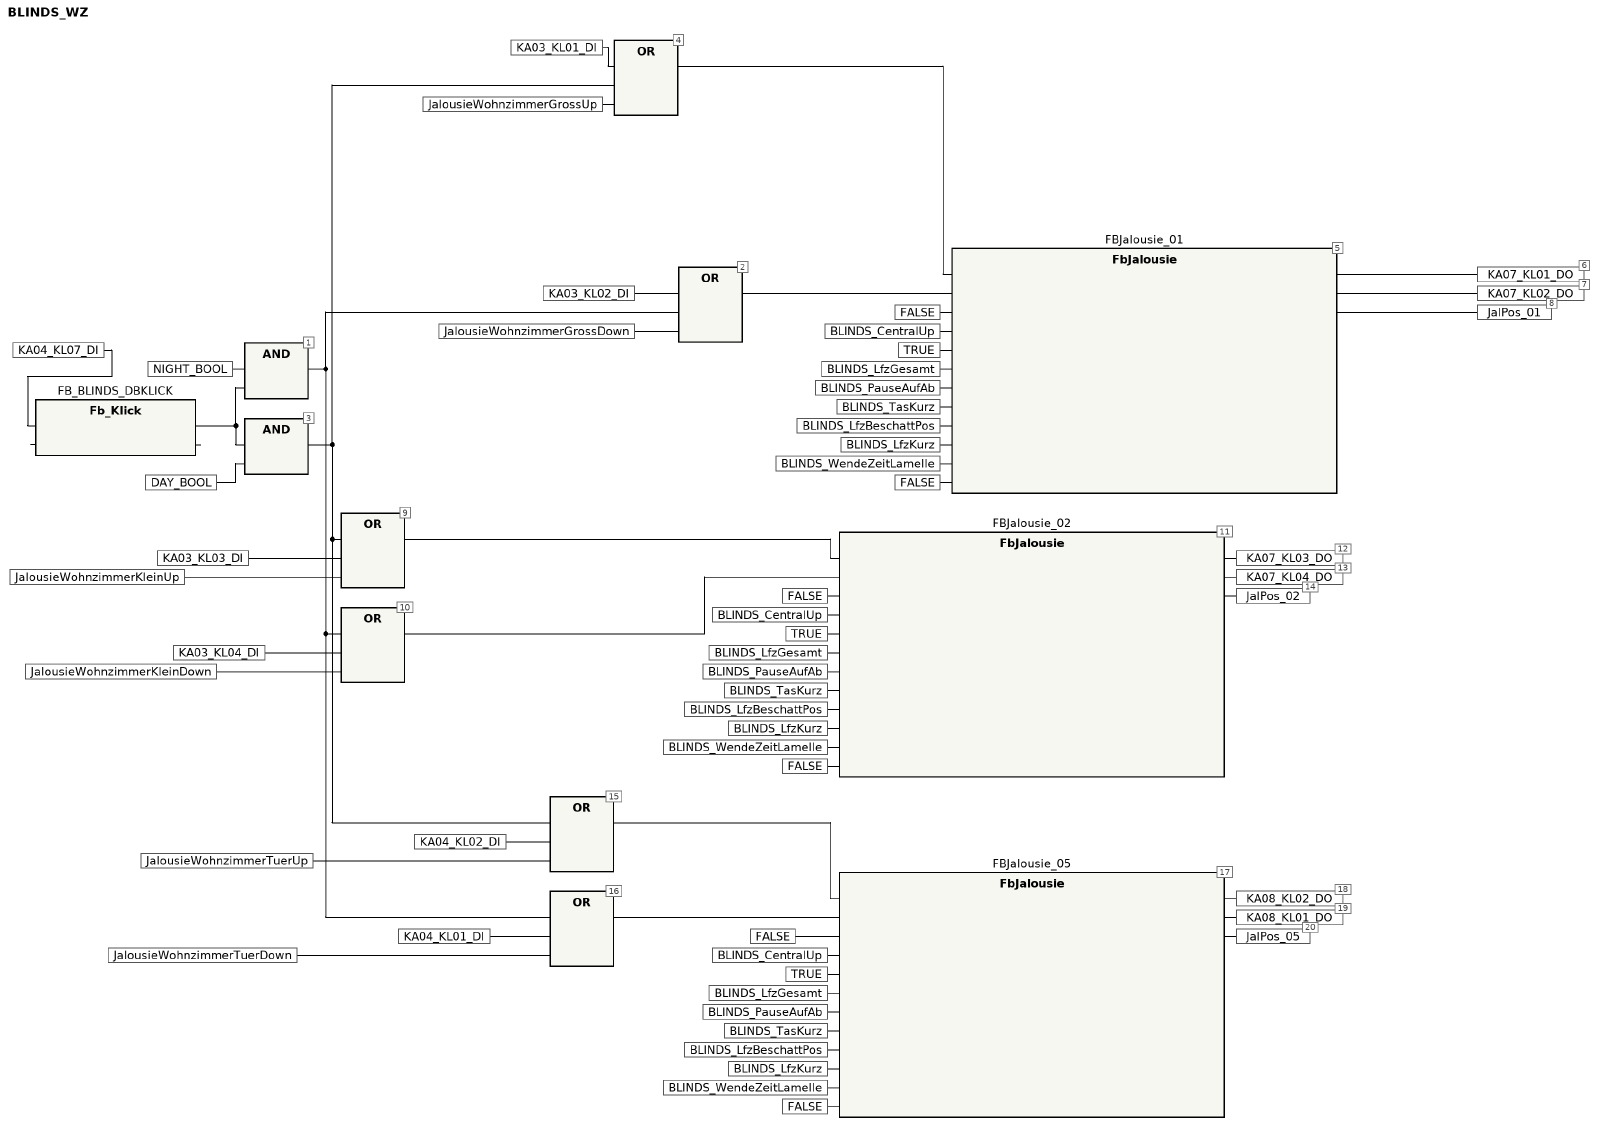
_CFC_ (* Continuous Function Chart, elements in execution order *)
#0 FB_BLINDS_DBKLICK:Fb_Klick(KA04_KL07_DI, -)
#1 AND(NIGHT_BOOL, #0.out 1)
#2 OR(KA03_KL02_DI, #1, JalousieWohnzimmerGrossDown)
#3 AND(#0.out 1, DAY_BOOL)
#4 OR(KA03_KL01_DI, #3, JalousieWohnzimmerGrossUp)
#5 FBJalousie_01:FbJalousie(#4, #2, FALSE, BLINDS_CentralUp, TRUE, BLINDS_LfzGesamt, BLINDS_PauseAufAb, BLINDS_TasKurz, BLINDS_LfzBeschattPos, BLINDS_LfzKurz, BLINDS_WendeZeitLamelle, FALSE)
#6 KA07_KL01_DO <= #5.out 1
#7 KA07_KL02_DO <= #5.out 2
#8 JalPos_01 <= #5.out 3
#9 OR(#3, KA03_KL03_DI, JalousieWohnzimmerKleinUp)
#10 OR(#1, KA03_KL04_DI, JalousieWohnzimmerKleinDown)
#11 FBJalousie_02:FbJalousie(#9, #10, FALSE, BLINDS_CentralUp, TRUE, BLINDS_LfzGesamt, BLINDS_PauseAufAb, BLINDS_TasKurz, BLINDS_LfzBeschattPos, BLINDS_LfzKurz, BLINDS_WendeZeitLamelle, FALSE)
#12 KA07_KL03_DO <= #11.out 1
#13 KA07_KL04_DO <= #11.out 2
#14 JalPos_02 <= #11.out 3
#15 OR(#3, KA04_KL02_DI, JalousieWohnzimmerTuerUp)
#16 OR(#1, KA04_KL01_DI, JalousieWohnzimmerTuerDown)
#17 FBJalousie_05:FbJalousie(#15, #16, FALSE, BLINDS_CentralUp, TRUE, BLINDS_LfzGesamt, BLINDS_PauseAufAb, BLINDS_TasKurz, BLINDS_LfzBeschattPos, BLINDS_LfzKurz, BLINDS_WendeZeitLamelle, FALSE)
#18 KA08_KL02_DO <= #17.out 1
#19 KA08_KL01_DO <= #17.out 2
#20 JalPos_05 <= #17.out 3
_END_CFC_
END_PROGRAM

(* POU BLINDS_ANNIKA, CFC *)
PROGRAM BLINDS_ANNIKA
VAR
	FBJalousie_03: FbJalousie;
	JalPos_03: BYTE;
END_VAR
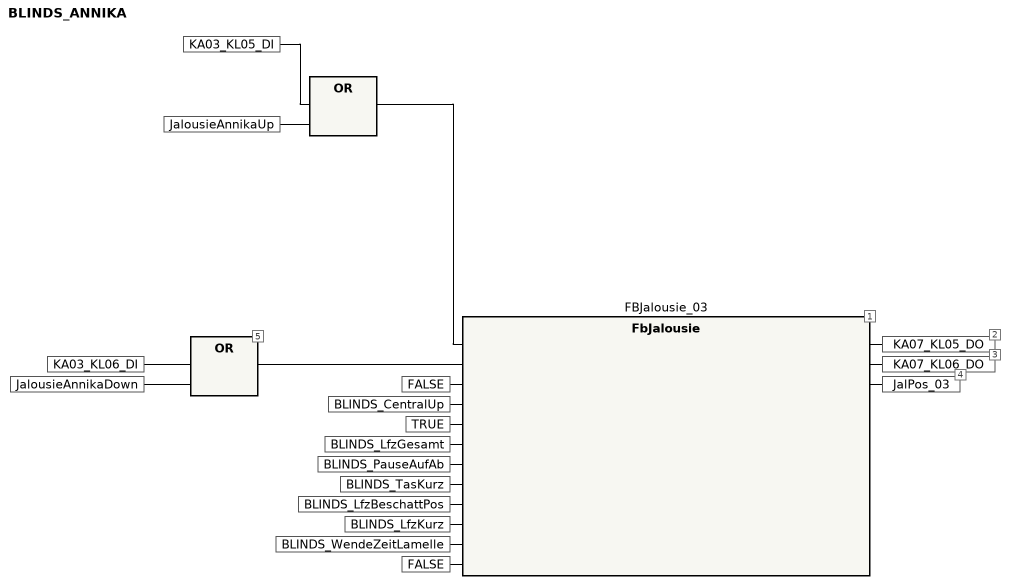
_CFC_ (* Continuous Function Chart, elements in execution order *)
#0 OR(KA03_KL05_DI, JalousieAnnikaUp)
#1 FBJalousie_03:FbJalousie(#0, #5, FALSE, BLINDS_CentralUp, TRUE, BLINDS_LfzGesamt, BLINDS_PauseAufAb, BLINDS_TasKurz, BLINDS_LfzBeschattPos, BLINDS_LfzKurz, BLINDS_WendeZeitLamelle, FALSE)
#2 KA07_KL05_DO <= #1.out 1
#3 KA07_KL06_DO <= #1.out 2
#4 JalPos_03 <= #1.out 3
#5 OR(KA03_KL06_DI, JalousieAnnikaDown)
_END_CFC_
END_PROGRAM

(* POU BLINDS_ELTERN, CFC *)
PROGRAM BLINDS_ELTERN
VAR
	FBJalousie_04: FbJalousie;
	JalPos_04: BYTE;

	R_TRIG_ElternUp_openhab: R_TRIG;
	F_TRIG_ElternUp_openhab: F_TRIG;
	Fb_Strmostooss_JalousieElternDown_openhab: Fb_Stromstoss;
	Fb_Stromstooss_JalousieElternUp_openhab: Fb_Stromstoss;
	R_TRIG_JalousieElternDown: R_TRIG;
	F_TRIG_JalousieElternDown: F_TRIG;
END_VAR
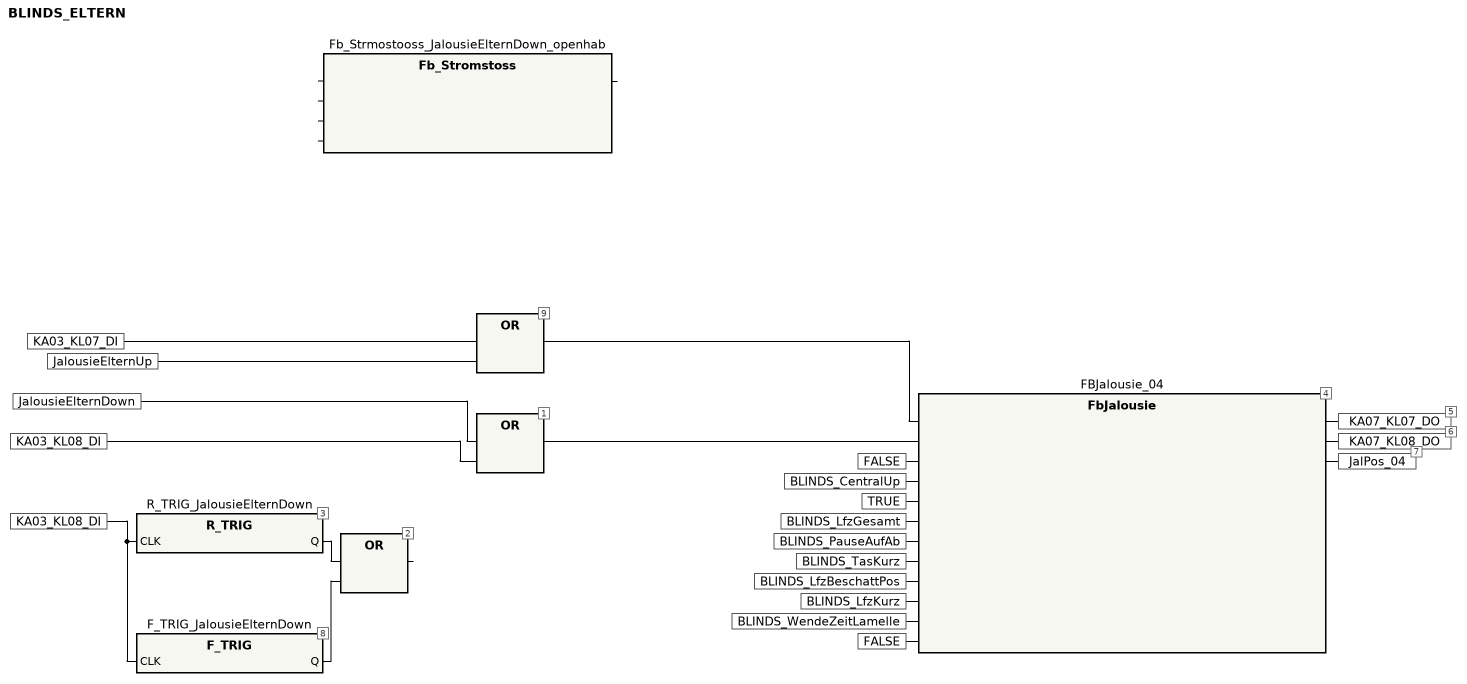
_CFC_ (* Continuous Function Chart, elements in execution order *)
#0 Fb_Strmostooss_JalousieElternDown_openhab:Fb_Stromstoss(-, -, -, -)
#1 OR(JalousieElternDown, KA03_KL08_DI)
#2 OR(#3.Q, #8.Q)
#3 R_TRIG_JalousieElternDown:R_TRIG(CLK: KA03_KL08_DI)
#4 FBJalousie_04:FbJalousie(#9, #1, FALSE, BLINDS_CentralUp, TRUE, BLINDS_LfzGesamt, BLINDS_PauseAufAb, BLINDS_TasKurz, BLINDS_LfzBeschattPos, BLINDS_LfzKurz, BLINDS_WendeZeitLamelle, FALSE)
#5 KA07_KL07_DO <= #4.out 1
#6 KA07_KL08_DO <= #4.out 2
#7 JalPos_04 <= #4.out 3
#8 F_TRIG_JalousieElternDown:F_TRIG(CLK: KA03_KL08_DI)
#9 OR(KA03_KL07_DI, JalousieElternUp)
_END_CFC_
END_PROGRAM

(* POU BLINDS_BUERO, CFC *)
PROGRAM BLINDS_BUERO
VAR
	FBJalousie_04: FbJalousie;
	JalPos_04: BYTE;

	R_TRIG_ElternUp_openhab: R_TRIG;
	F_TRIG_ElternUp_openhab: F_TRIG;
	Fb_Strmostooss_JalousieElternDown_openhab: Fb_Stromstoss;
	Fb_Stromstooss_JalousieElternUp_openhab: Fb_Stromstoss;
	R_TRIG_JalousieElternDown: R_TRIG;
	F_TRIG_JalousieElternDown: F_TRIG;
END_VAR
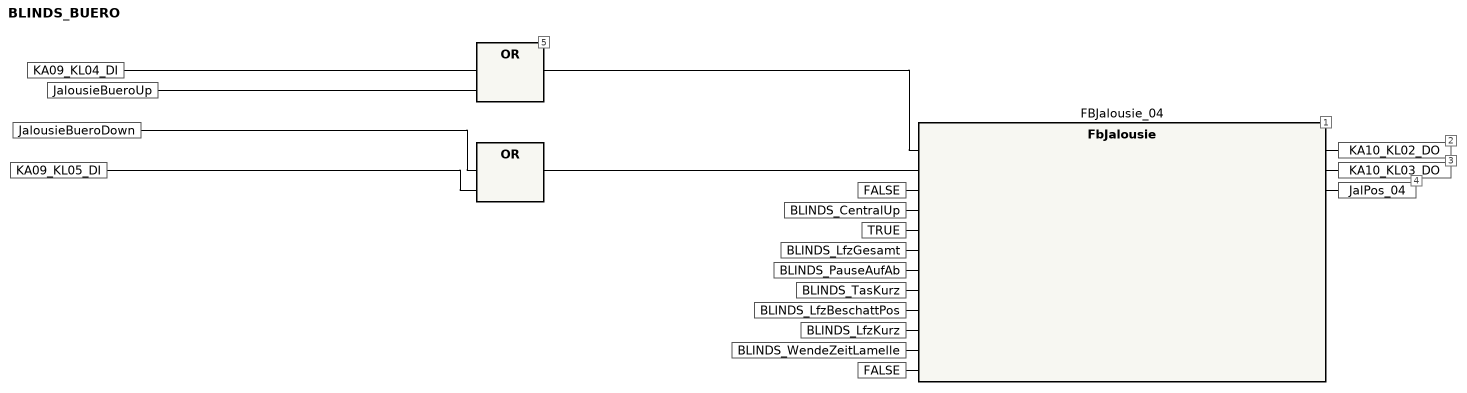
_CFC_ (* Continuous Function Chart, elements in execution order *)
#0 OR(JalousieBueroDown, KA09_KL05_DI)
#1 FBJalousie_04:FbJalousie(#5, #0, FALSE, BLINDS_CentralUp, TRUE, BLINDS_LfzGesamt, BLINDS_PauseAufAb, BLINDS_TasKurz, BLINDS_LfzBeschattPos, BLINDS_LfzKurz, BLINDS_WendeZeitLamelle, FALSE)
#2 KA10_KL02_DO <= #1.out 1
#3 KA10_KL03_DO <= #1.out 2
#4 JalPos_04 <= #1.out 3
#5 OR(KA09_KL04_DI, JalousieBueroUp)
_END_CFC_
END_PROGRAM

(* POU BLINDS_KUECHE, CFC *)
PROGRAM BLINDS_KUECHE
VAR
	FBJalousie_04: FbJalousie;
	JalPos_04: BYTE;

	R_TRIG_ElternUp_openhab: R_TRIG;
	F_TRIG_ElternUp_openhab: F_TRIG;
	Fb_Strmostooss_JalousieElternDown_openhab: Fb_Stromstoss;
	Fb_Stromstooss_JalousieElternUp_openhab: Fb_Stromstoss;
	R_TRIG_JalousieElternDown: R_TRIG;
	F_TRIG_JalousieElternDown: F_TRIG;
	JalousieBueroUp: BOOL;
      JalousieBueroDown: BOOL;
END_VAR
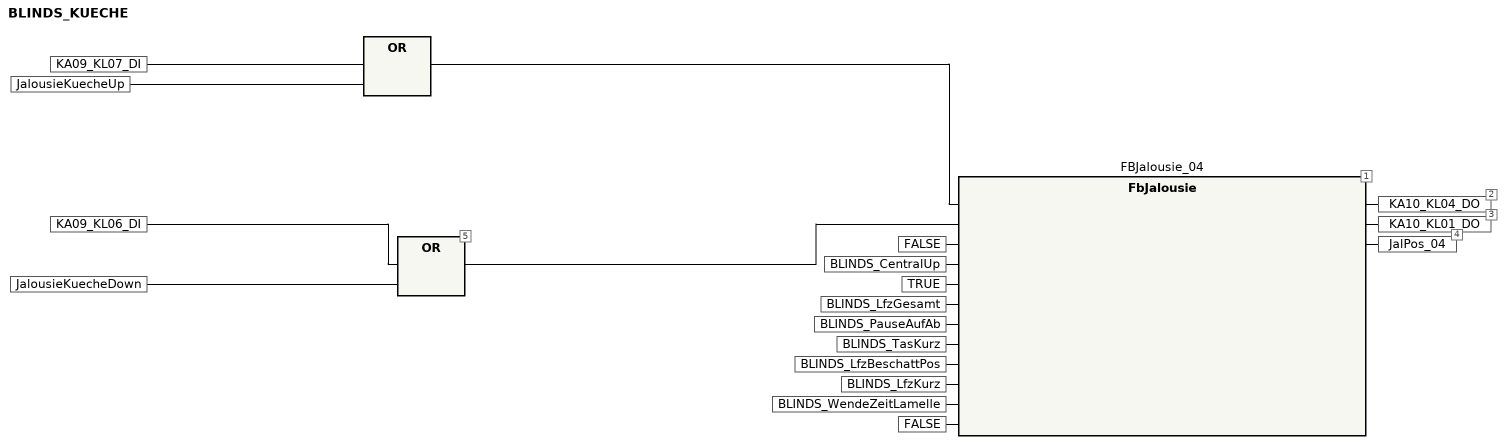
_CFC_ (* Continuous Function Chart, elements in execution order *)
#0 OR(KA09_KL07_DI, JalousieKuecheUp)
#1 FBJalousie_04:FbJalousie(#0, #5, FALSE, BLINDS_CentralUp, TRUE, BLINDS_LfzGesamt, BLINDS_PauseAufAb, BLINDS_TasKurz, BLINDS_LfzBeschattPos, BLINDS_LfzKurz, BLINDS_WendeZeitLamelle, FALSE)
#2 KA10_KL04_DO <= #1.out 1
#3 KA10_KL01_DO <= #1.out 2
#4 JalPos_04 <= #1.out 3
#5 OR(KA09_KL06_DI, JalousieKuecheDown)
_END_CFC_
END_PROGRAM

(* POU LIGHTS_ATTIC, CFC *)
PROGRAM LIGHTS_ATTIC
VAR
	R_TRIG_ATTIC_1: R_TRIG;
	F_TRIG_ATTIC_1: F_TRIG;
	FB_LIGHT_ATTIC_1: FbLatchedRelay;
	Fb_KurzLang: Fb_KurzLang;
	FB_LIGHT_ATTIC_2: FbLatchedRelay;
	Fb_Klick_Attic_1: Fb_Klick;
	R_TRIG_DACHBODEN_openhab: R_TRIG;
	F_TRIG_DACHBODEN_openhab: F_TRIG;
END_VAR
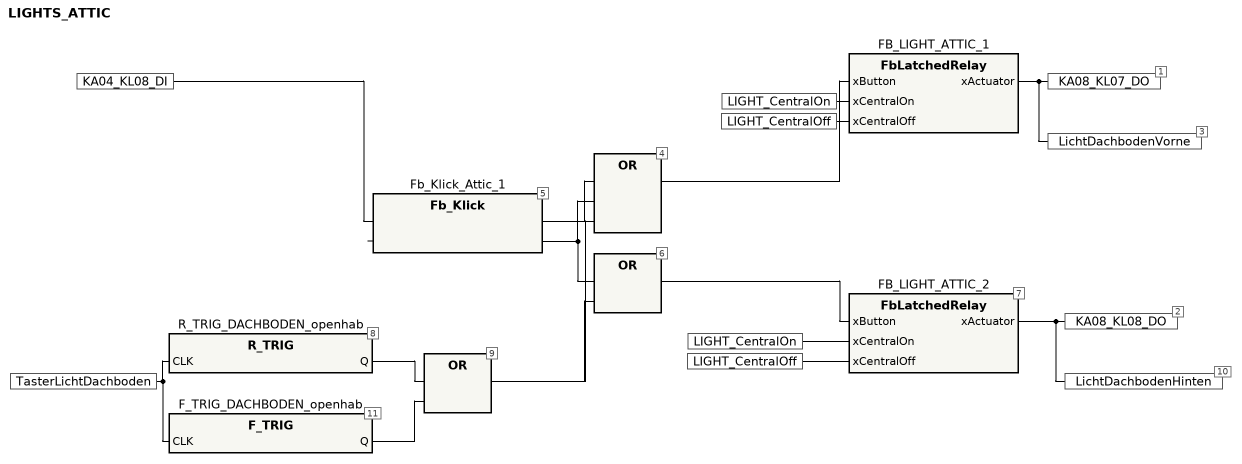
_CFC_ (* Continuous Function Chart, elements in execution order *)
#0 FB_LIGHT_ATTIC_1:FbLatchedRelay(xButton: #4, xCentralOn: LIGHT_CentralOn, xCentralOff: LIGHT_CentralOff)
#1 KA08_KL07_DO <= #0.xActuator
#2 KA08_KL08_DO <= #7.xActuator
#3 LichtDachbodenVorne <= #0.xActuator
#4 OR(#5.out 1, #5.out 2, #9)
#5 Fb_Klick_Attic_1:Fb_Klick(KA04_KL08_DI, -)
#6 OR(#5.out 2, #9)
#7 FB_LIGHT_ATTIC_2:FbLatchedRelay(xButton: #6, xCentralOn: LIGHT_CentralOn, xCentralOff: LIGHT_CentralOff)
#8 R_TRIG_DACHBODEN_openhab:R_TRIG(CLK: TasterLichtDachboden)
#9 OR(#8.Q, #11.Q)
#10 LichtDachbodenHinten <= #7.xActuator
#11 F_TRIG_DACHBODEN_openhab:F_TRIG(CLK: TasterLichtDachboden)
_END_CFC_
END_PROGRAM

(* POU IsDay, ST *)
PROGRAM IsDay
VAR
	MyDateTime: DT;
	MyTime: TIME;
	myTime2: SysTime64;
END_VAR
IF HOUR > 18 OR HOUR < 5 THEN
	NIGHT_BOOL := TRUE;
	DAY_BOOL := FALSE;
ELSE
       NIGHT_BOOL := FALSE;
	DAY_BOOL := TRUE;
END_IF


MyDateTime := SysRtcGetTime(TRUE);
MyTime := DT_TO_TIME(MyDateTime);
END_PROGRAM

(* POU BLINDS, CFC *)
PROGRAM BLINDS
VAR
	FBJalousie_01: FbJalousie;
	JalPos_01: BYTE;
	FBJalousie_02: FbJalousie;
	JalPos_02: BYTE;
	FBJalousie_05: FbJalousie;
	JalPos_05: BYTE;

END_VAR
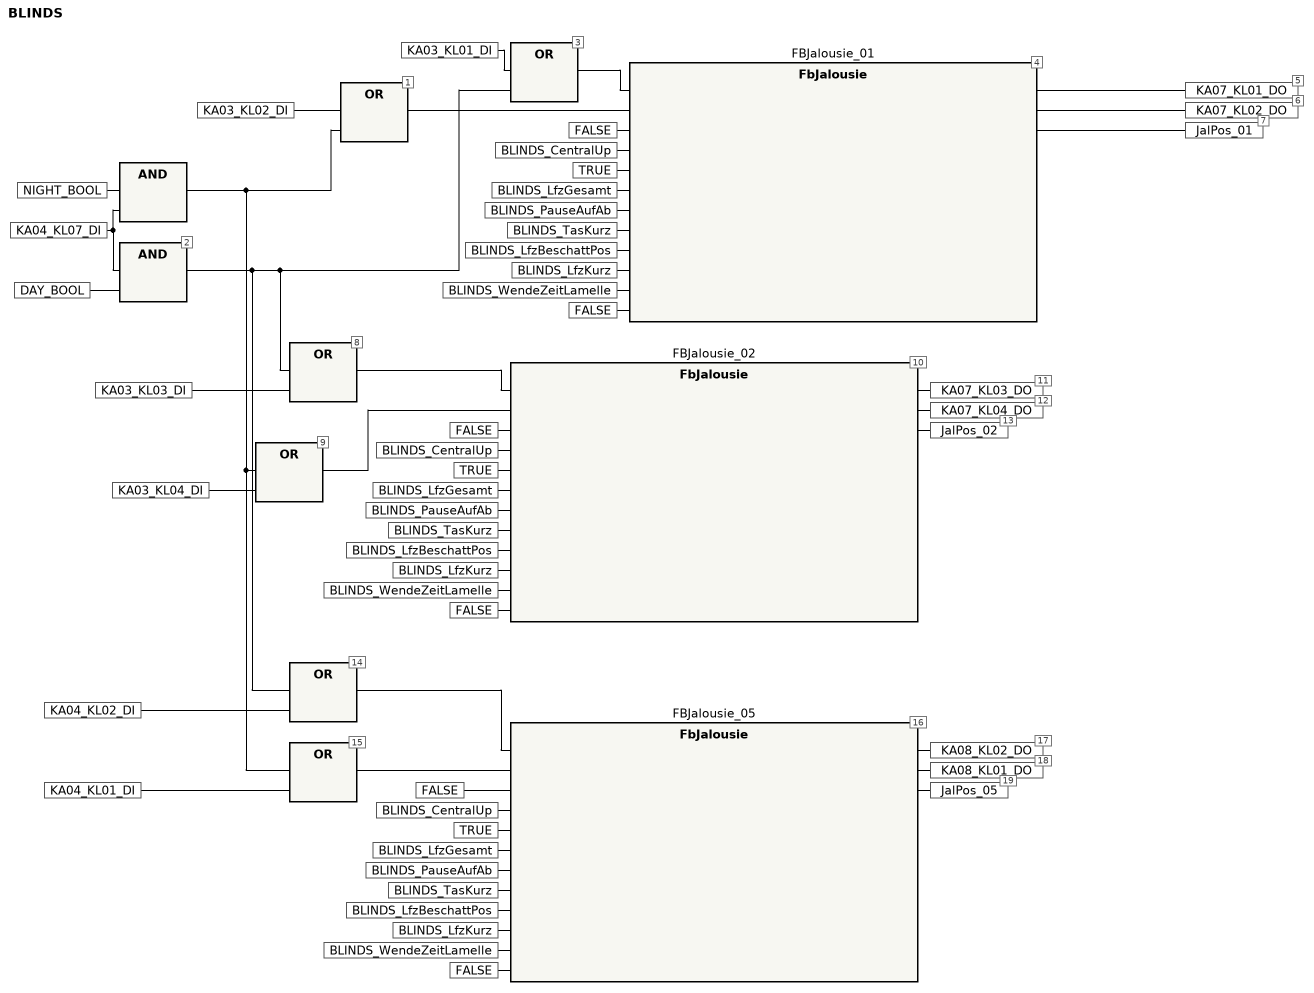
_CFC_ (* Continuous Function Chart, elements in execution order *)
#0 AND(NIGHT_BOOL, KA04_KL07_DI)
#1 OR(KA03_KL02_DI, #0)
#2 AND(KA04_KL07_DI, DAY_BOOL)
#3 OR(KA03_KL01_DI, #2)
#4 FBJalousie_01:FbJalousie(#3, #1, FALSE, BLINDS_CentralUp, TRUE, BLINDS_LfzGesamt, BLINDS_PauseAufAb, BLINDS_TasKurz, BLINDS_LfzBeschattPos, BLINDS_LfzKurz, BLINDS_WendeZeitLamelle, FALSE)
#5 KA07_KL01_DO <= #4.out 1
#6 KA07_KL02_DO <= #4.out 2
#7 JalPos_01 <= #4.out 3
#8 OR(#2, KA03_KL03_DI)
#9 OR(#0, KA03_KL04_DI)
#10 FBJalousie_02:FbJalousie(#8, #9, FALSE, BLINDS_CentralUp, TRUE, BLINDS_LfzGesamt, BLINDS_PauseAufAb, BLINDS_TasKurz, BLINDS_LfzBeschattPos, BLINDS_LfzKurz, BLINDS_WendeZeitLamelle, FALSE)
#11 KA07_KL03_DO <= #10.out 1
#12 KA07_KL04_DO <= #10.out 2
#13 JalPos_02 <= #10.out 3
#14 OR(#2, KA04_KL02_DI)
#15 OR(#0, KA04_KL01_DI)
#16 FBJalousie_05:FbJalousie(#14, #15, FALSE, BLINDS_CentralUp, TRUE, BLINDS_LfzGesamt, BLINDS_PauseAufAb, BLINDS_TasKurz, BLINDS_LfzBeschattPos, BLINDS_LfzKurz, BLINDS_WendeZeitLamelle, FALSE)
#17 KA08_KL02_DO <= #16.out 1
#18 KA08_KL01_DO <= #16.out 2
#19 JalPos_05 <= #16.out 3
_END_CFC_
END_PROGRAM

(* POU Configuration/MODBUS_CONFIGURATION, ST *)
PROGRAM MODBUS_CONFIGURATION
VAR                                
END_VAR                            
(*                                 
   <?xml version="1.0" encoding="UTF-16" standalone="yes"?>
<network xml_structure_version="1" xml_feature_version="1">
	<generator_settings minRTUTaskCycleTimeMs="5" minEthaskCycleTimeMs="5" ethSlaveMultiplier="0.1" rtuInterfaceMultiplier="0.1" taskGeneration="true"/>
</network>
                              
*)                                 
;                                  
END_PROGRAM
